// TIA Portal V19 export
DATA_BLOCK "Area0301_V_Counter_IDB"   // DB62
// stored: InstanceOfName VirtualEncoder, InstanceOfType FB
"VirtualEncoder"
   // VAR_INPUT
   //    ActualSpeed : LReal;
   //    OB_Cycle : UDInt;
   // END_VAR
   // VAR_IN_OUT
   //    VCounter : LReal;
   // END_VAR
   // VAR
   //    InitDone : Bool;
   //    ActualSpeed_mm_s : LReal;
   //    PrevSpeed_mm_s : LReal;
   //    DeltaT_s : LReal;
   //    DeltaV : LReal;
   //    DeltaS : LReal;
   // END_VAR
BEGIN
END_DATA_BLOCK
